// Mitsubishi GX Works2 project: guide_kommunikasjon_slave   PLC: FX3U/FX3UC

// global labels: Global1
VAR_GLOBAL
  lampe_0 AT Y000 : BOOL;
  lampe_1 AT Y001 : BOOL;
  lampeVar_0 AT M100 : BOOL;
  lampeVar_1 AT M101 : BOOL;
  anaDig AT D8260 : INT;
  digAna AT D8262 : INT;
  slider AT D0 : INT;
  tank AT D1 : INT;
END_VAR

// task Task_01 (event TRUE, interval 0, priority 31): POU_01

PROGRAM POU_01
(* structured ladder/FBD written out as ST: instructions are called as NAME(EN, inputs, outputs); _pN, _eN, _tN stand for wires *)
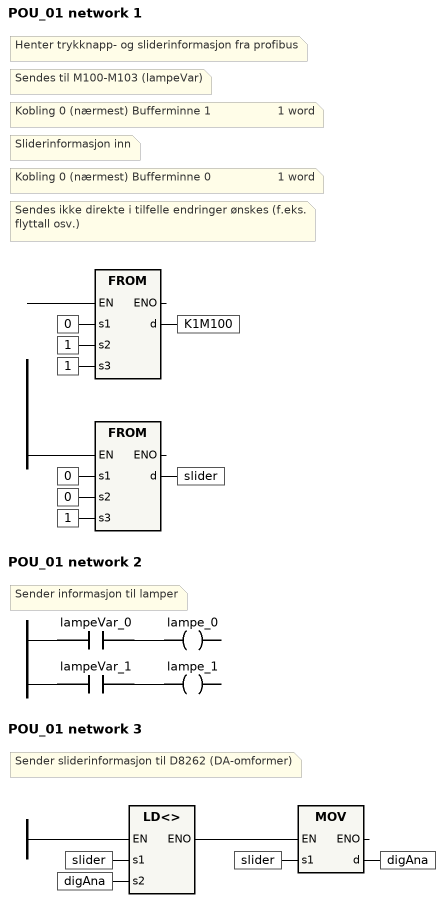
(* network 1 *)
(* Henter trykknapp- og sliderinformasjon fra profibus *)
(* Sendes til M100-M103 (lampeVar) *)
(* Kobling 0 (nærmest) Bufferminne 1                   1 word *)
(* Sliderinformasjon inn *)
(* Kobling 0 (nærmest) Bufferminne 0                   1 word *)
(* Sendes ikke direkte i tilfelle endringer ønskes (f.eks. flyttall osv.) *)
FROM(TRUE, 0, 1, 1, K1M100);
FROM(TRUE, 0, 0, 1, slider);
(* network 2 *)
(* Sender informasjon til lamper *)
lampe_0 := lampeVar_0;
lampe_1 := lampeVar_1;
(* network 3 *)
(* Sender sliderinformasjon til D8262 (DA-omformer) *)
_e1 := LD<>(TRUE, slider, digAna);
MOV(_e1, slider, digAna);
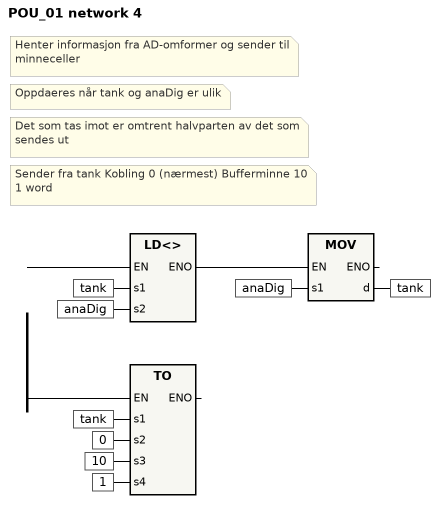
(* network 4 *)
(* Henter informasjon fra AD-omformer og sender til minneceller *)
(* Oppdaeres når tank og anaDig er ulik *)
(* Det som tas imot er omtrent halvparten av det som sendes ut *)
(* Sender fra tank Kobling 0 (nærmest) Bufferminne 10           1 word *)
_e1 := LD<>(TRUE, tank, anaDig);
MOV(_e1, anaDig, tank);
TO(TRUE, tank, 0, 10, 1);
END_PROGRAM
